(* CODESYS project PrviZadatak.project
   CustomField04_name: CustomField04
   CustomField06_name: CustomField06
   CustomField07_name: CustomField07
   CustomField09_name: CustomField09
   CustomField08_name: CustomField08
   CustomField02_name: CustomField02
   CustomField10_name: CustomField10
   CustomField01_name: CustomField01
   CustomField03_name: CustomField03
   CustomField05_name: CustomField05

Project tree, tasks and I/O mapping:
  MyController : TM238LFDC24DT, Schneider Electric, order no. TM238LFDC24DT, version 2.0.31.8
    application Application
      task MAST (cyclic, interval 20 ms, priority 15, watchdog 100 ms x 1) calls POU_LADDER
      global variables GVL
      function HiddenPOU [ST]
      program POU_LADDER [LD]
    CAN
    Serial Line 1
      Modbus_Manager : Modbus_Manager, Schneider Electric, version 2.0.1.12
    Embedded Functions
      IO : IO, Schneider Electric, version 2.0.31.8
          input  Application.POU_LADDER.Tipkalo2 : BOOL  // IW0.I9
          input  Application.POU_LADDER.Tipkalo1 : BOOL  // IW0.I10
          input  Application.POU_LADDER.Sklopka1 : BOOL  // IW0.I11
          input  Application.POU_LADDER.Sklopka2 : BOOL  // IW0.I12
          output Application.POU_LADDER.Zelena1 : BOOL  // QW0.Q4
          output Application.POU_LADDER.Zuta1 : BOOL  // QW0.Q5
          output Application.POU_LADDER.Crvena1 : BOOL  // QW0.Q6
          output Application.POU_LADDER.Zelena2 : BOOL  // QW0.Q7
          output Application.POU_LADDER.Zuta2 : BOOL  // QW0.Q8
          output Application.POU_LADDER.Crvena2 : BOOL  // QW0.Q9
          unmapped channels: IW0, QW0
      HSC : HSC, Schneider Electric, version 2.0.31.8
        HSC
      PTO_PWM : PTO_PWM, Schneider Electric, version 2.0.31.8
        PTO_PWM
    Serial Line 2
      SoMachine_Network_Manager : SoMachine-Network_Manager, Schneider Electric, version 2.0.1.10
  MachineLayoutPicture
*)

// MyController/Application/GVL
VAR_GLOBAL
END_VAR

// MyController/Application/POU_LADDER
PROGRAM POU_LADDER
VAR
	Sklopka1: BOOL;
	Sklopka2: BOOL;
	Tipkalo1: BOOL;
	Zelena1: BOOL;
	Tipkalo2: BOOL;
	Crvena1: BOOL;
	Crvena2: BOOL;
	Zelena2: BOOL;
	Zuta1: BOOL;
	Zuta2: BOOL;
END_VAR
VAR // added by the converter: edge detectors and wires of the graphical bodies
    _w1 : BOOL;
END_VAR

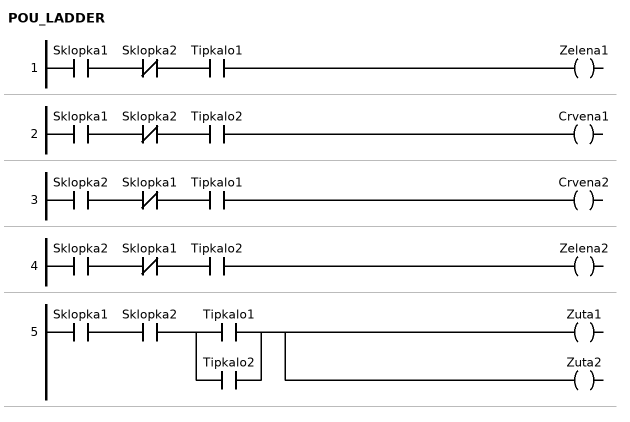
// NETWORK 1
Zelena1 := Sklopka1 AND NOT Sklopka2 AND Tipkalo1;

// NETWORK 2
Crvena1 := Sklopka1 AND NOT Sklopka2 AND Tipkalo2;

// NETWORK 3
Crvena2 := Sklopka2 AND NOT Sklopka1 AND Tipkalo1;

// NETWORK 4
Zelena2 := Sklopka2 AND NOT Sklopka1 AND Tipkalo2;

// NETWORK 5
_w1 := Sklopka1 AND Sklopka2 AND (Tipkalo1 OR Tipkalo2);
Zuta1 := _w1;
Zuta2 := _w1;

END_PROGRAM

// MyController/Application/HiddenPOU
FUNCTION HiddenPOU : BOOL

VAR_INPUT
	pHiddenFunc: POINTER TO WORD;
END_VAR
VAR
	pRead: POINTER TO BYTE;
	pWrite: POINTER TO BYTE;
END_VAR

pRead := pHiddenFunc + 400;
pWrite := pHiddenFunc + 4400;
HiddenPOU := TRUE;

END_FUNCTION
